PROGRAM MAIN
VAR
END_VAR

END_PROGRAM

(* stored: Version 1.1.0.1
   POU MAIN: Id {82ccea0c-f4b1-4f8c-852a-ee292c7f124e} *)
